FUNCTION_BLOCK FB_Timer
VAR
	fb_tonTimer:TON;
	tTime: TIME;
	tTimeMid: TIME;
	uiTime:UINT;
END_VAR

METHOD init : BOOL
tTimeMid:=T#0S;
fb_tonTimer(IN :=0);
END_METHOD

METHOD timer : BOOL
VAR_INPUT
	bStart: BOOL;
END_VAR
VAR_OUTPUT
	uiTimeHour: UINT;
	uiTimeMinute: UINT;
	uiTimeSecond: UINT;
END_VAR
fb_tonTimer(IN:=bStart, PT:=T#999H , );
IF NOT fb_tonTimer.IN THEN
	tTimeMid:=tTime;
END_IF	

tTime:=fb_tonTimer.ET+tTimeMid;
uiTime:=DT_TO_UINT(TIME_TO_DT(tTime));
uiTimeHour:= uiTime/3600;
uiTimeMinute:= uiTime/60-uiTimeHour*60;
uiTimeSecond:= uiTime-uiTimeHour*3600-uiTimeMinute*60;
END_METHOD

END_FUNCTION_BLOCK

(* stored: Version 1.1.0.1, ProductVersion 3.1.4024.11
   POU FB_Timer: Id {2554a4c0-5698-48c5-b7c9-8d2fdf4902b6}, SpecialFunc None
   Method init: Id {3da09fc7-d006-4917-ab67-a69425b55ec6}
   Method timer: Id {e7de819b-88b0-457f-aef0-60c24077759c} *)
